FUNCTION_BLOCK FB_LinearActuator EXTENDS FB_StateMachine  IMPLEMENTS I_StateMachine
VAR_INPUT
	bStartHoming : BOOL;
	bEnable : BOOL;
	bStartJog : BOOL;
	bStartHalt : BOOL;
	bStartStop : BOOL;
	
END_VAR
VAR
	eInnerState : E_LinearActuatorStates;
	fbHoming	: FB_LinearActuatorHoming;
	stAxis		: ST_LinearActuatorAxis;
END_VAR

OuterLopSM();

METHOD Disable : BOOL

VAR
	bChildBusy  : BOOL := FALSE;
END_VAR
fbHoming(bActive:=FALSE);



IF fbHoming.Busy THEN
	bChildBusy := TRUE;
ELSIF fbHoming.bError THEN
	bChildBusy := TRUE;
	{warning 'TODO: trigger e-stop'}
	//	Stack trace and bError switching are reserved for inner loop
	fbHoming.ErrorAck:=TRUE;
END_IF



IF bChildBusy THEN
	Disable := FALSE;
ELSE
	Disable := TRUE;
END_IF
END_METHOD

PROPERTY ForceHoming : BOOL
GET
ForceHoming := stAxis.bForceHoming;
END_GET
SET
stAxis.bForceHoming := ForceHoming;
END_SET
END_PROPERTY

PROPERTY Homed : BOOL
GET
IF bActive THEN
	Homed := NOT fbHoming.HomingNeeded;
ELSE
	Homed :=  TRUE;;
END_IF
END_GET
END_PROPERTY

METHOD InnerLoopSM : BOOL
// update all children FBs
fbHoming();

CASE CyclicInnerCase(TO_STRING(eInnerState)) OF
	E_LinearActuatorStates.Idle:
		IF bStartHoming THEN
			bStartHoming := FALSE;
			ChangeInnerState(E_LinearActuatorStates.Homing1);
		END_IF

	E_LinearActuatorStates.Homing1:
		IF fbHoming.Busy THEN
			// fbHoming should never be busy here 	
			sErrorDetails := 'fbHoming.Busy = TRUE';
			fbEventHandler(eNapID:=E_Event.UNABLE_TO_START_TASK,sMessage:=sErrorDetails);
			bError := TRUE;	
		ELSE
			IF fbHoming.bError THEN
				sErrorDetails := 'fbHoming.bReady=FALSE';
				fbEventHandler(eNapID:=E_Event.UNABLE_TO_START_TASK,sMessage:=sErrorDetails);
				bError := TRUE;
			ELSE
				fbHoming.bStart:=TRUE;
				ChangeInnerState(E_LinearActuatorStates.Homing2);
			END_IF
		END_IF
		
		
	E_LinearActuatorStates.Homing2:
		IF fbHoming.Busy THEN
			// Wait... fbStepper still busy 			
		ELSE
			IF fbHoming.bError THEN
				fbEventHandler(eNapID:=E_Event.TASK_FAILED,sTrace:=fbHoming.EventTrace);
				fbHoming.ErrorAck:=TRUE;
				bError := TRUE;
			ELSE
				IF Homed THEN
					fbEventHandler(eNapID:=E_Event.REQUEST_COMPLETED);
					ChangeInnerState(E_LinearActuatorStates.Idle);
				ELSE
					sErrorDetails := 'Homed=FALSE';
					fbEventHandler(eNapID:=E_Event.TASK_FAILED,sMessage:=sErrorDetails);
					bError := TRUE;
				END_IF
			END_IF
		END_IF
END_CASE
END_METHOD

PROPERTY Position : LREAL
GET
Position := stAxis.stAxisRef.NcToPlc.ActPos;
END_GET
END_PROPERTY

METHOD PUBLIC ReadStatus : BOOL
stAxis.stAxisRef.ReadStatus();
{warning 'TODO: add logit to update stAxis.bAtTopPosition'}
END_METHOD

METHOD Reset : BOOL
// reset variables specific to this FB 

// Reactivate children FBs
fbHoming.Active:=TRUE;
END_METHOD

METHOD Setup : BOOL
eStateMachineSourceID := eStateSourceID;
fbHoming(eStateSourceID := THIS^.eStateMachineSourceID +  E_LinearActuatorID_Offset.LinearActuatorHoming,
					aErrorLog:=THIS^.aErrorLog,
					nErrorLogIndex:=THIS^.nErrorLogIndex,
					stParentsAxis:=THIS^.stAxis);
					
SetInnerEnumeration(nStateEnum:=THIS^.eInnerState);
END_METHOD

END_FUNCTION_BLOCK

(* stored: Version 1.1.0.1, ProductVersion 3.1.4024.12
   POU FB_LinearActuator: Id {39ffc351-0f6a-4f95-915f-ef1e54ac00b2}, SpecialFunc None
   Folder Properties: Id {67b8ba1b-0009-4384-9a87-257fa03c62cd}
   Method Disable: Id {2c1f58b5-63e4-4bb8-9cf0-e61d1c2de641}
   Property ForceHoming: Id {98c0a965-5128-4826-9949-f56fb5be7ee0}
   Get Get: Id {cdd72a7a-0011-4c9b-b322-e9b5b64592d1}
   Set Set: Id {b4ef3e88-69c5-48c2-bef5-fae65f7e1168}
   Property Homed: Id {6cc8ab12-d7db-47a9-8164-075c35a1b665}
   Get Get: Id {e14a833a-2065-4add-8a1d-e8399fbcf4b0}
   Method InnerLoopSM: Id {35781a01-7cb5-4d9c-9a89-3e2cef93d299}
   Property Position: Id {db193924-7987-4438-959b-5229a7c4f28b}
   Get Get: Id {254a0463-4f21-4d81-9ebd-cd167752e5fd}
   Method ReadStatus: Id {ed33bb7d-4920-4997-b14d-20e2decde0a3}
   Method Reset: Id {99379e88-438c-4b03-8a4e-ced232c5b93d}
   Method Setup: Id {20854eb8-c628-493a-b732-db16588a4af4} *)
